// TIA Portal V19 export
FUNCTION_BLOCK "MonitoringValves"   // FB1, STL
{ S7_Optimized_Access := 'TRUE' }
// stored: AutoNumber false, MemoryReserve 100
   VAR
      V01_01 : "ValveMonitor";
      V01_03 : "ValveMonitor";
      V01_04 : "ValveMonitor";
      V01_08 : "ValveMonitor";
      V01_09 : "ValveMonitor";
      V01_11 : "ValveMonitor";
      V01_12 : "ValveMonitor";
      V01_13 : "ValveMonitor";
      V01_14 : "ValveMonitor";
      V01_15 : "ValveMonitor";
      V01_16 : "ValveMonitor";
      V01_17 : "ValveMonitor";
      V09_01 : "ValveMonitor";
      V09_02 : "ValveMonitor";
      V09_03 : "ValveMonitor";
      V09_04 : "ValveMonitor";
      V09_05 : "ValveMonitor";
      V09_06 : "ValveMonitor";
      V09_07 : "ValveMonitor";
      V09_08 : "ValveMonitor";
      V09_09 : "ValveMonitor";
      V09_10 : "ValveMonitor";
      V09_11 : "ValveMonitor";
      V09_12 : "ValveMonitor";
   END_VAR
   VAR_TEMP
      DoubleFB : Word;
      En_Only : Word;
      De_Only : Word;
   END_VAR
BEGIN

NETWORK
TITLE = 
      L     16#0300;
      T     #DoubleFB;
      L     16#0200;
      T     #De_Only;
      L     16#0100;
      T     #En_Only;



      CALL  #V01_01
      ( IN_EN       := "Y0101S",  // Energised Feedback input
        IN_DE       := "Y0101R",  // De-Energised Feedback input
        IN_ACT      := "Y0101",
        ControlWord := #DoubleFB,
        Info        := "ValvesScadaInfo".V01_01  // SCADA Interface
      );



      CALL  #V01_03
      ( IN_EN       := "Y0103S",
        IN_DE       := "Y0103R",
        IN_ACT      := "Y0103",
        ControlWord := #DoubleFB,
        Info        := "ValvesScadaInfo".V01_03
      );

      CALL  #V01_04
      ( IN_EN       := "Y0104S",
        IN_DE       := "Y0104R",
        IN_ACT      := "Y0104",
        ControlWord := #DoubleFB,
        Info        := "ValvesScadaInfo".V01_04
      );

      CALL  #V01_08
      ( IN_EN       := "Y0108S",
        IN_DE       := "Y0108R",
        IN_ACT      := "Y0108",
        ControlWord := #DoubleFB,
        Info        := "ValvesScadaInfo".V01_08
      );

      CALL  #V01_09
      ( IN_EN       := "Y0109S",
        IN_DE       := "Y0109R",
        IN_ACT      := "Y0109",
        ControlWord := #DoubleFB,
        Info        := "ValvesScadaInfo".V01_09
      );

      CALL  #V01_11
      ( IN_EN       := "Y0111S",
        IN_DE       := "Y0111R",
        IN_ACT      := "Y0111",
        ControlWord := #DoubleFB,
        Info        := "ValvesScadaInfo".V01_11
      );


      CALL  #V01_12
      ( IN_EN       := "Y0112S",
        IN_DE       := "Y0112R",
        IN_ACT      := "Y0112",
        ControlWord := #DoubleFB,
        Info        := "ValvesScadaInfo".V01_12
      );

      CALL  #V01_13
      ( IN_EN       := "Y0113S",
        IN_DE       := "Y0113R",
        IN_ACT      := "Y0113",
        ControlWord := #DoubleFB,
        Info        := "ValvesScadaInfo".V01_13
      );

      CALL  #V01_14
      ( IN_EN       := "Y0114S",
        IN_DE       := "Y0114R",
        IN_ACT      := "Y0114",
        ControlWord := #DoubleFB,
        Info        := "ValvesScadaInfo".V01_14
      );


      CALL  #V01_15
      ( IN_EN       := "Y0115S",
        IN_DE       := "Y0115R",
        IN_ACT      := "Y0115",
        ControlWord := #DoubleFB,
        Info        := "ValvesScadaInfo".V01_15
      );

      CALL  #V01_16
      ( IN_EN       := "Y0116S",
        IN_DE       := "Y0116R",
        IN_ACT      := "Y0116",
        ControlWord := #DoubleFB,
        Info        := "ValvesScadaInfo".V01_16
      );

      CALL  #V01_17
      ( IN_EN       := "Y0117S",
        IN_DE       := "Y0117R",
        IN_ACT      := "Y0117",
        ControlWord := #DoubleFB,
        Info        := "ValvesScadaInfo".V01_17
      );



      CALL  #V09_04
      ( IN_EN       := "Y0904S",
        IN_DE       := "Y0904R",
        IN_ACT      := "Y0904",
        ControlWord := #DoubleFB,
        Info        := "ValvesScadaInfo".V09_04
      );


      CALL  #V09_05
      ( IN_EN       := "Y0905S",
        IN_DE       := "Y0905R",
        IN_ACT      := "Y0905",
        ControlWord := #DoubleFB,
        Info        := "ValvesScadaInfo".V09_05
      );

      CALL  #V09_06
      ( IN_EN       := "Y0906S",
        IN_DE       := "Y0906R",
        IN_ACT      := "Y0906",
        ControlWord := #DoubleFB,
        Info        := "ValvesScadaInfo".V09_06
      );

      CALL  #V09_07
      ( IN_EN       := "Y0907S",
        IN_DE       := "Y0907R",
        IN_ACT      := "Y0907",
        ControlWord := #DoubleFB,
        Info        := "ValvesScadaInfo".V09_07
      );

      CALL  #V09_08
      ( IN_EN       := "Y0908S",
        IN_DE       := "Y0908R",
        IN_ACT      := "Y0908",
        ControlWord := #DoubleFB,
        Info        := "ValvesScadaInfo".V09_08
      );

      CALL  #V09_09
      ( IN_EN       := "Y0909S",
        IN_DE       := "Y0909R",
        IN_ACT      := "Y0909",
        ControlWord := #DoubleFB,
        Info        := "ValvesScadaInfo".V09_09
      );

      CALL  #V09_10
      ( IN_EN       := "Y0910S",
        IN_DE       := "Y0910R",
        IN_ACT      := "Y0910",
        ControlWord := #DoubleFB,
        Info        := "ValvesScadaInfo".V09_10
      );


      CALL  #V09_11
      ( IN_EN       := "Y0911S",
        IN_DE       := "Y0911R",
        IN_ACT      := "Y0911",
        ControlWord := #DoubleFB,
        Info        := "ValvesScadaInfo".V09_11
      );


      CALL  #V09_12
      ( IN_EN       := "Y0912S",
        IN_DE       := "Y0912R",
        IN_ACT      := "Y0912",
        ControlWord := #DoubleFB,
        Info        := "ValvesScadaInfo".V09_12
      );


END_FUNCTION_BLOCK
